# EPICS autosave request: iocBoot/ioc13lab2/auto_positions.req
file "CARS_8_motor_positions.req", P=13LAB2:
